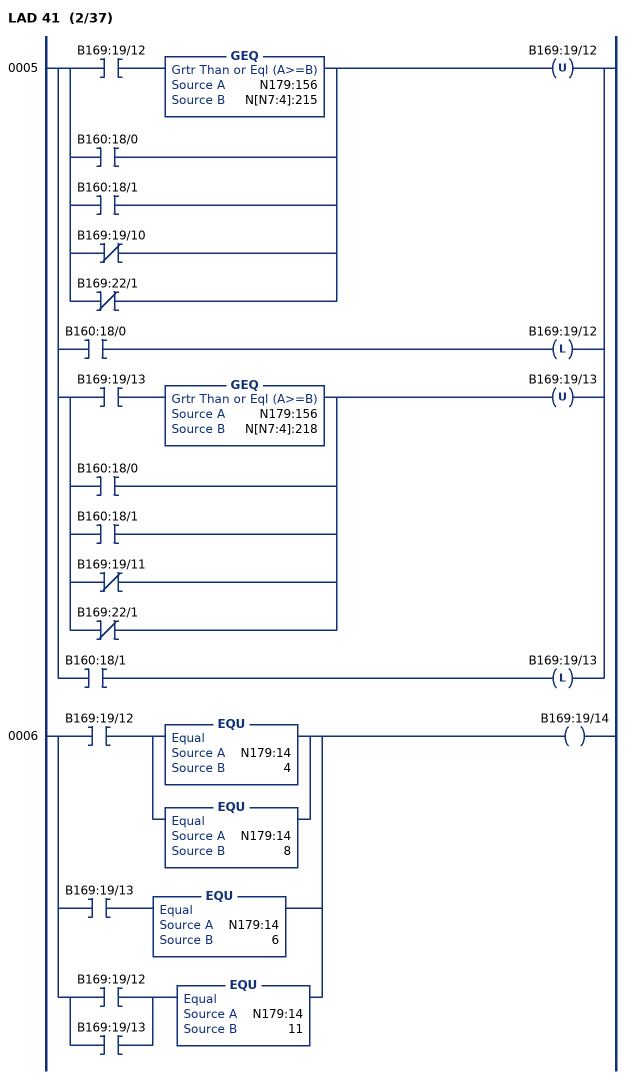
% Rung: 5 %
SOR BST BST BST XIC B169:19/12 GEQ N179:156 N[N7:4]:215 NXB BST XIC B160:18/0 NXB XIC B160:18/1 BND NXB XIO B169:19/10 NXB XIO B169:22/1 BND OTU B169:19/12 NXB XIC B160:18/0 OTL B169:19/12 BND NXB BST BST XIC B169:19/13 GEQ N179:156 N[N7:4]:218 NXB BST XIC B160:18/0 NXB XIC B160:18/1 BND NXB XIO B169:19/11 NXB XIO B169:22/1 BND OTU B169:19/13 NXB XIC B160:18/1 OTL B169:19/13 BND BND EOR
% Rung: 6 %
SOR BST XIC B169:19/12 BST EQU N179:14 4 NXB EQU N179:14 8 BND NXB XIC B169:19/13 EQU N179:14 6 NXB BST XIC B169:19/12 NXB XIC B169:19/13 BND EQU N179:14 11 BND OTE B169:19/14 EOR

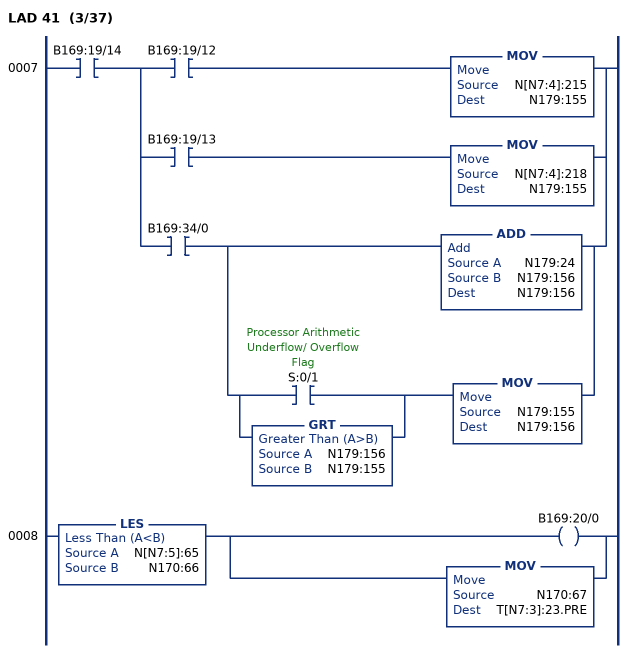
% Rung: 7 %
SOR XIC B169:19/14 BST BST XIC B169:19/12 MOV N[N7:4]:215 N179:155 NXB XIC B169:19/13 MOV N[N7:4]:218 N179:155 BND NXB XIC B169:34/0 BST ADD N179:24 N179:156 N179:156 NXB BST XIC S:0/1 NXB GRT N179:156 N179:155 BND MOV N179:155 N179:156 BND BND EOR
%   S:0/1  "Processor Arithmetic Underflow/ Overflow Flag" %
% Rung: 8 %
SOR LES N[N7:5]:65 N170:66 BST OTE B169:20/0 NXB MOV N170:67 T[N7:3]:23.PRE BND EOR

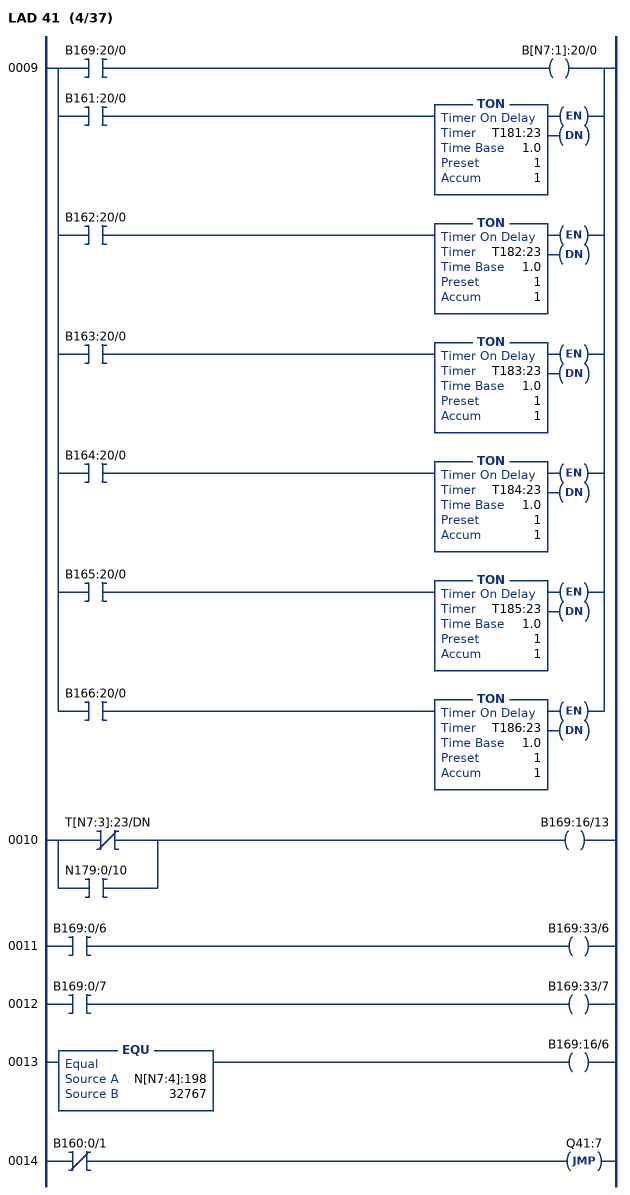
% Rung: 9 %
SOR BST XIC B169:20/0 OTE B[N7:1]:20/0 NXB XIC B161:20/0 TON T181:23 1.0 1 1 NXB XIC B162:20/0 TON T182:23 1.0 1 1 NXB XIC B163:20/0 TON T183:23 1.0 1 1 NXB XIC B164:20/0 TON T184:23 1.0 1 1 NXB XIC B165:20/0 TON T185:23 1.0 1 1 NXB XIC B166:20/0 TON T186:23 1.0 1 1 BND EOR
% Rung: 10 %
SOR BST XIO T[N7:3]:23/DN NXB XIC N179:0/10 BND OTE B169:16/13 EOR
% Rung: 11 %
SOR XIC B169:0/6 OTE B169:33/6 EOR
% Rung: 12 %
SOR XIC B169:0/7 OTE B169:33/7 EOR
% Rung: 13 %
SOR EQU N[N7:4]:198 32767 OTE B169:16/6 EOR
% Rung: 14 %
SOR XIO B160:0/1 JMP Q41:7 EOR

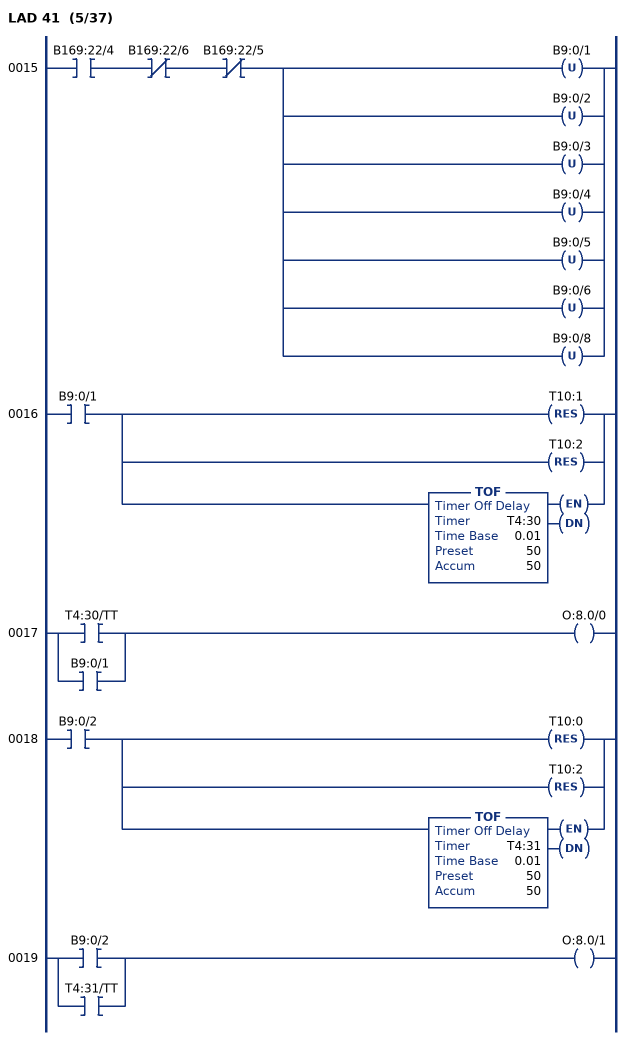
% Rung: 15 %
SOR XIC B169:22/4 XIO B169:22/6 XIO B169:22/5 BST OTU B9:0/1 NXB OTU B9:0/2 NXB OTU B9:0/3 NXB OTU B9:0/4 NXB OTU B9:0/5 NXB OTU B9:0/6 NXB OTU B9:0/8 BND EOR
% Rung: 16 %
SOR XIC B9:0/1 BST RES T10:1 NXB RES T10:2 NXB TOF T4:30 0.01 50 50 BND EOR
% Rung: 17 %
SOR BST XIC T4:30/TT NXB XIC B9:0/1 BND OTE O:8.0/0 EOR
% Rung: 18 %
SOR XIC B9:0/2 BST RES T10:0 NXB RES T10:2 NXB TOF T4:31 0.01 50 50 BND EOR
% Rung: 19 %
SOR BST XIC B9:0/2 NXB XIC T4:31/TT BND OTE O:8.0/1 EOR

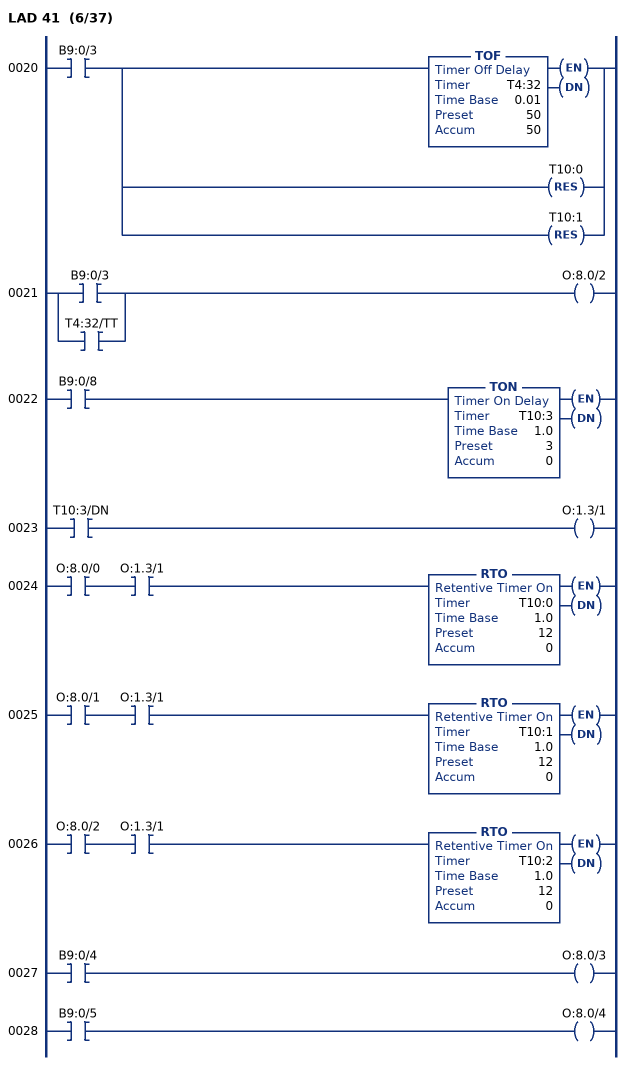
% Rung: 20 %
SOR XIC B9:0/3 BST TOF T4:32 0.01 50 50 NXB RES T10:0 NXB RES T10:1 BND EOR
% Rung: 21 %
SOR BST XIC B9:0/3 NXB XIC T4:32/TT BND OTE O:8.0/2 EOR
% Rung: 22 %
SOR XIC B9:0/8 TON T10:3 1.0 3 0 EOR
% Rung: 23 %
SOR XIC T10:3/DN OTE O:1.3/1 EOR
% Rung: 24 %
SOR XIC O:8.0/0 XIC O:1.3/1 RTO T10:0 1.0 12 0 EOR
% Rung: 25 %
SOR XIC O:8.0/1 XIC O:1.3/1 RTO T10:1 1.0 12 0 EOR
% Rung: 26 %
SOR XIC O:8.0/2 XIC O:1.3/1 RTO T10:2 1.0 12 0 EOR
% Rung: 27 %
SOR XIC B9:0/4 OTE O:8.0/3 EOR
% Rung: 28 %
SOR XIC B9:0/5 OTE O:8.0/4 EOR

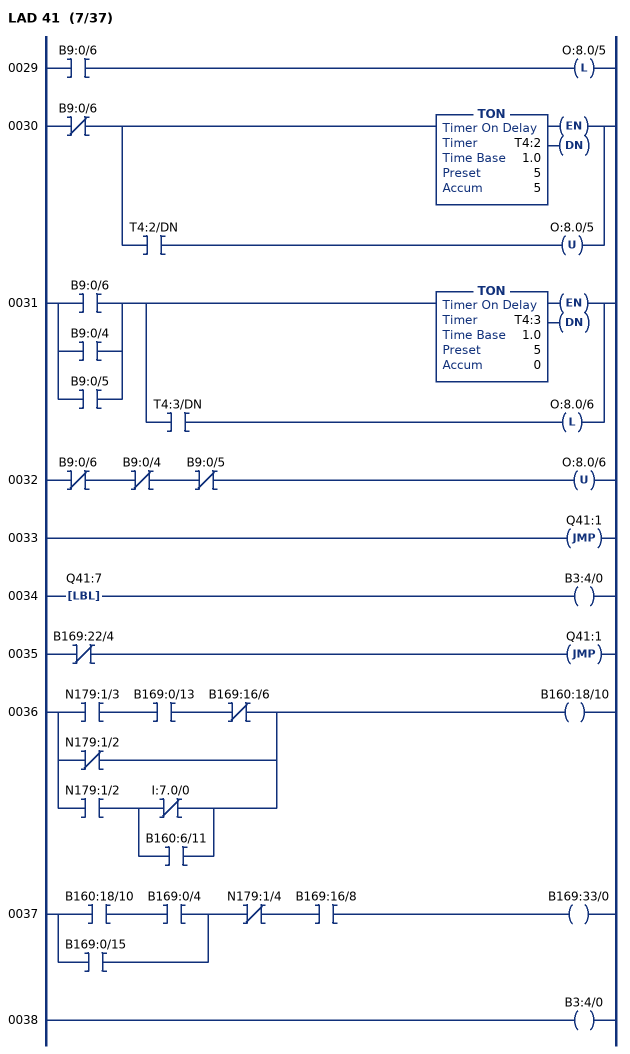
% Rung: 29 %
SOR XIC B9:0/6 OTL O:8.0/5 EOR
% Rung: 30 %
SOR XIO B9:0/6 BST TON T4:2 1.0 5 5 NXB XIC T4:2/DN OTU O:8.0/5 BND EOR
% Rung: 31 %
SOR BST XIC B9:0/6 NXB BST XIC B9:0/4 NXB XIC B9:0/5 BND BND BST TON T4:3 1.0 5 0 NXB XIC T4:3/DN OTL O:8.0/6 BND EOR
% Rung: 32 %
SOR XIO B9:0/6 XIO B9:0/4 XIO B9:0/5 OTU O:8.0/6 EOR
% Rung: 33 %
SOR JMP Q41:1 EOR
% Rung: 34 %
SOR LBL Q41:7 OTE B3:4/0 EOR
% Rung: 35 %
SOR XIO B169:22/4 JMP Q41:1 EOR
% Rung: 36 %
SOR BST XIC N179:1/3 XIC B169:0/13 XIO B169:16/6 NXB XIO N179:1/2 NXB XIC N179:1/2 BST XIO I:7.0/0 NXB XIC B160:6/11 BND BND OTE B160:18/10 EOR
% Rung: 37 %
SOR BST XIC B160:18/10 XIC B169:0/4 NXB XIC B169:0/15 BND XIO N179:1/4 XIC B169:16/8 OTE B169:33/0 EOR
% Rung: 38 %
SOR OTE B3:4/0 EOR

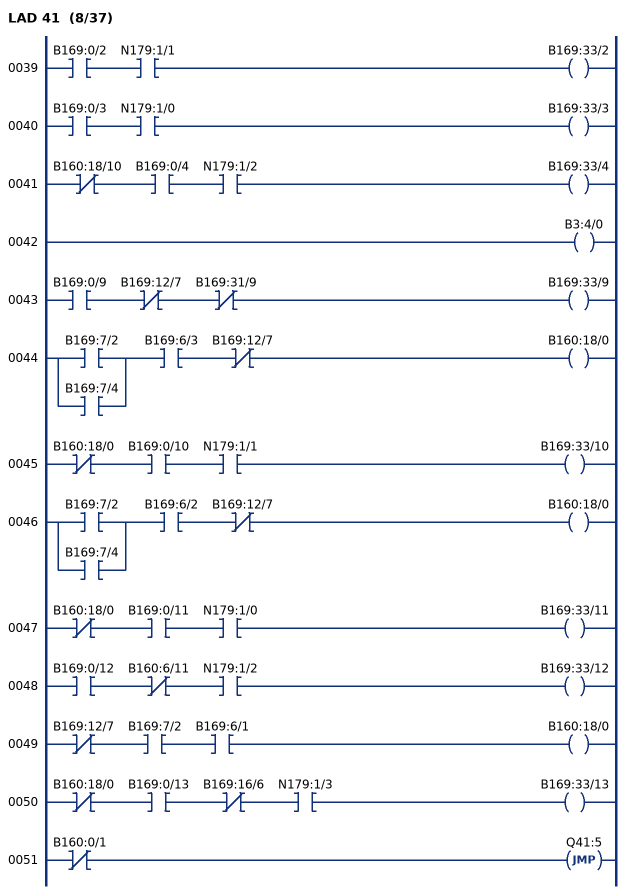
% Rung: 39 %
SOR XIC B169:0/2 XIC N179:1/1 OTE B169:33/2 EOR
% Rung: 40 %
SOR XIC B169:0/3 XIC N179:1/0 OTE B169:33/3 EOR
% Rung: 41 %
SOR XIO B160:18/10 XIC B169:0/4 XIC N179:1/2 OTE B169:33/4 EOR
% Rung: 42 %
SOR OTE B3:4/0 EOR
% Rung: 43 %
SOR XIC B169:0/9 XIO B169:12/7 XIO B169:31/9 OTE B169:33/9 EOR
% Rung: 44 %
SOR BST XIC B169:7/2 NXB XIC B169:7/4 BND XIC B169:6/3 XIO B169:12/7 OTE B160:18/0 EOR
% Rung: 45 %
SOR XIO B160:18/0 XIC B169:0/10 XIC N179:1/1 OTE B169:33/10 EOR
% Rung: 46 %
SOR BST XIC B169:7/2 NXB XIC B169:7/4 BND XIC B169:6/2 XIO B169:12/7 OTE B160:18/0 EOR
% Rung: 47 %
SOR XIO B160:18/0 XIC B169:0/11 XIC N179:1/0 OTE B169:33/11 EOR
% Rung: 48 %
SOR XIC B169:0/12 XIO B160:6/11 XIC N179:1/2 OTE B169:33/12 EOR
% Rung: 49 %
SOR XIO B169:12/7 XIC B169:7/2 XIC B169:6/1 OTE B160:18/0 EOR
% Rung: 50 %
SOR XIO B160:18/0 XIC B169:0/13 XIO B169:16/6 XIC N179:1/3 OTE B169:33/13 EOR
% Rung: 51 %
SOR XIO B160:0/1 JMP Q41:5 EOR

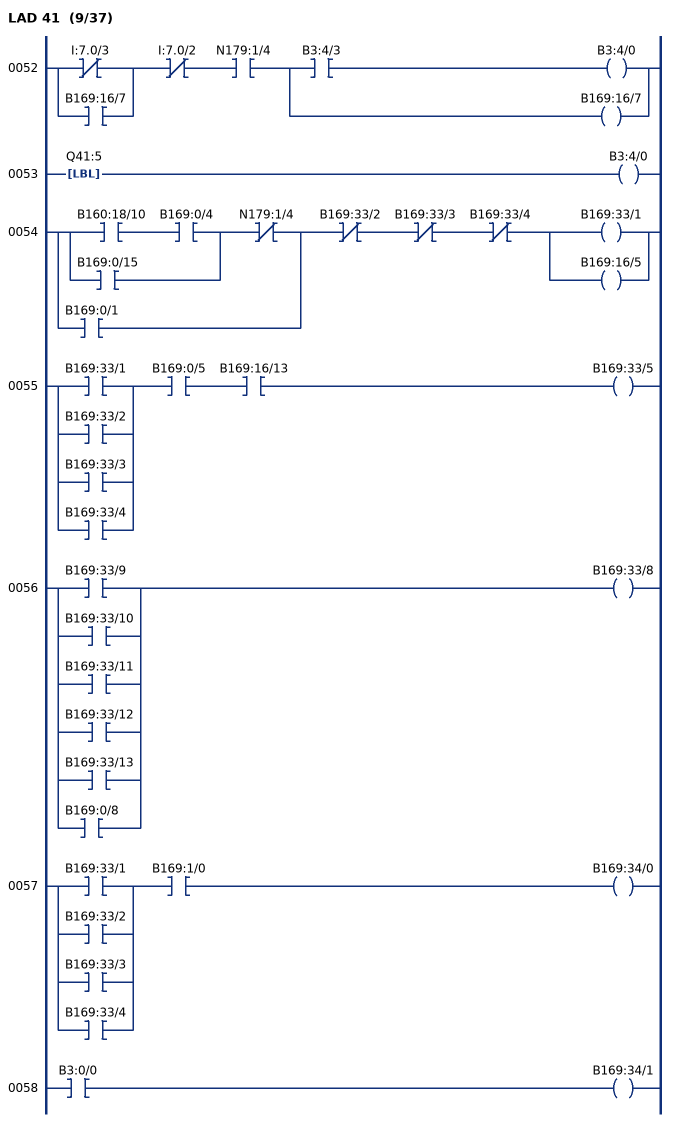
% Rung: 52 %
SOR BST XIO I:7.0/3 NXB XIC B169:16/7 BND XIO I:7.0/2 XIC N179:1/4 BST XIC B3:4/3 OTE B3:4/0 NXB OTE B169:16/7 BND EOR
% Rung: 53 %
SOR LBL Q41:5 OTE B3:4/0 EOR
% Rung: 54 %
SOR BST BST XIC B160:18/10 XIC B169:0/4 NXB XIC B169:0/15 BND XIO N179:1/4 NXB XIC B169:0/1 BND XIO B169:33/2 XIO B169:33/3 XIO B169:33/4 BST OTE B169:33/1 NXB OTE B169:16/5 BND EOR
% Rung: 55 %
SOR BST XIC B169:33/1 NXB XIC B169:33/2 NXB XIC B169:33/3 NXB XIC B169:33/4 BND XIC B169:0/5 XIC B169:16/13 OTE B169:33/5 EOR
% Rung: 56 %
SOR BST XIC B169:33/9 NXB XIC B169:33/10 NXB XIC B169:33/11 NXB XIC B169:33/12 NXB XIC B169:33/13 NXB XIC B169:0/8 BND OTE B169:33/8 EOR
% Rung: 57 %
SOR BST XIC B169:33/1 NXB XIC B169:33/2 NXB XIC B169:33/3 NXB XIC B169:33/4 BND XIC B169:1/0 OTE B169:34/0 EOR
% Rung: 58 %
SOR XIC B3:0/0 OTE B169:34/1 EOR

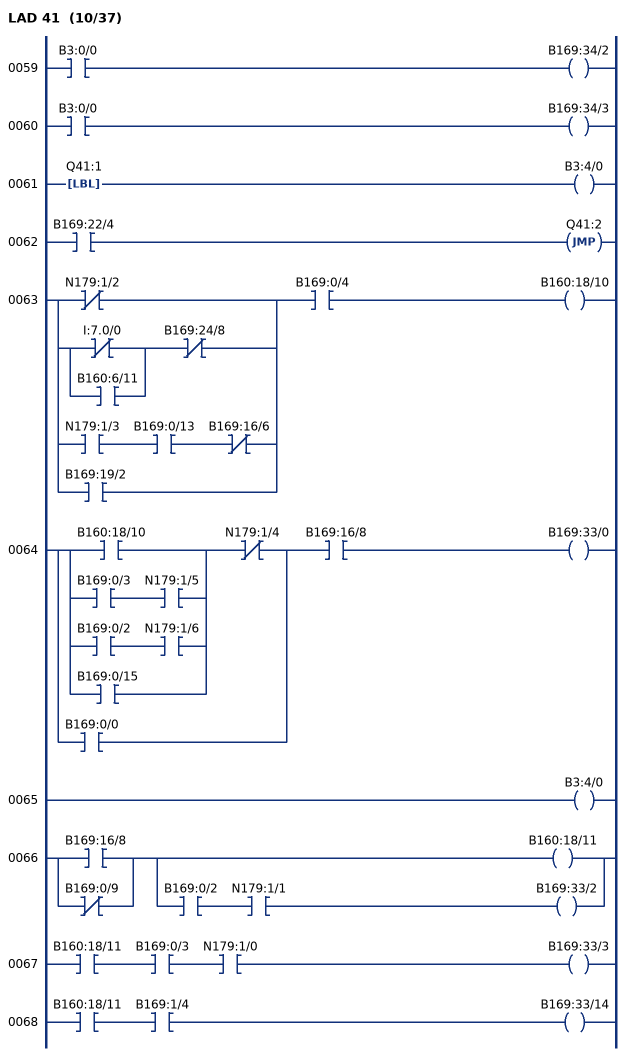
% Rung: 59 %
SOR XIC B3:0/0 OTE B169:34/2 EOR
% Rung: 60 %
SOR XIC B3:0/0 OTE B169:34/3 EOR
% Rung: 61 %
SOR LBL Q41:1 OTE B3:4/0 EOR
% Rung: 62 %
SOR XIC B169:22/4 JMP Q41:2 EOR
% Rung: 63 %
SOR BST XIO N179:1/2 NXB BST XIO I:7.0/0 NXB XIC B160:6/11 BND XIO B169:24/8 NXB XIC N179:1/3 XIC B169:0/13 XIO B169:16/6 NXB XIC B169:19/2 BND XIC B169:0/4 OTE B160:18/10 EOR
% Rung: 64 %
SOR BST BST XIC B160:18/10 NXB XIC B169:0/3 XIC N179:1/5 NXB XIC B169:0/2 XIC N179:1/6 NXB XIC B169:0/15 BND XIO N179:1/4 NXB XIC B169:0/0 BND XIC B169:16/8 OTE B169:33/0 EOR
% Rung: 65 %
SOR OTE B3:4/0 EOR
% Rung: 66 %
SOR BST XIC B169:16/8 NXB XIO B169:0/9 BND BST OTE B160:18/11 NXB XIC B169:0/2 XIC N179:1/1 OTE B169:33/2 BND EOR
% Rung: 67 %
SOR XIC B160:18/11 XIC B169:0/3 XIC N179:1/0 OTE B169:33/3 EOR
% Rung: 68 %
SOR XIC B160:18/11 XIC B169:1/4 OTE B169:33/14 EOR

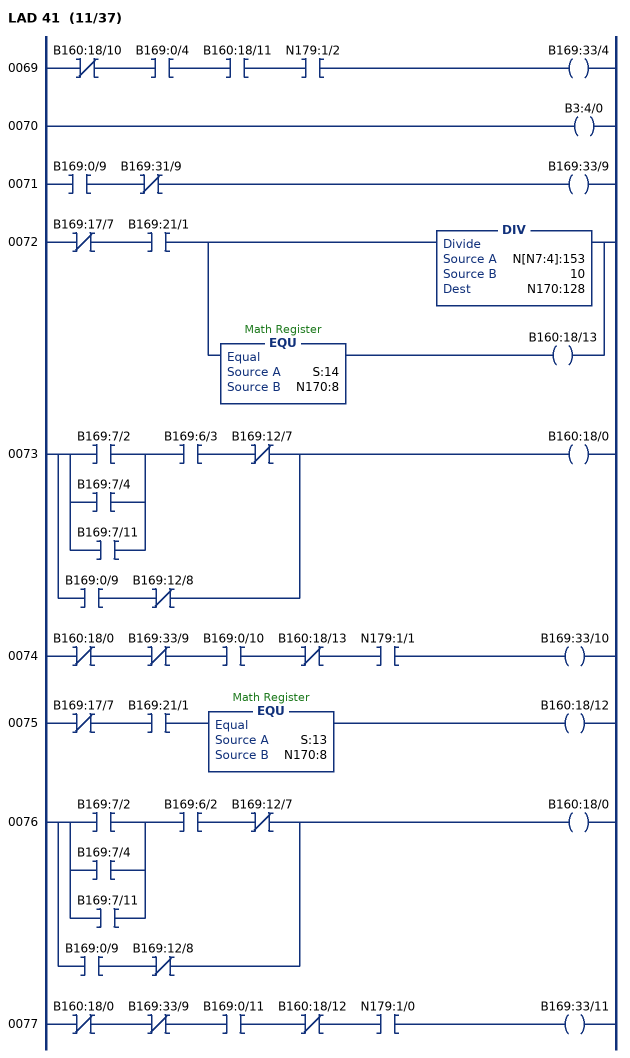
% Rung: 69 %
SOR XIO B160:18/10 XIC B169:0/4 XIC B160:18/11 XIC N179:1/2 OTE B169:33/4 EOR
% Rung: 70 %
SOR OTE B3:4/0 EOR
% Rung: 71 %
SOR XIC B169:0/9 XIO B169:31/9 OTE B169:33/9 EOR
% Rung: 72 %
SOR XIO B169:17/7 XIC B169:21/1 BST DIV N[N7:4]:153 10 N170:128 NXB EQU S:14 N170:8 OTE B160:18/13 BND EOR
%   S:14  "Math Register" %
% Rung: 73 %
SOR BST BST XIC B169:7/2 NXB XIC B169:7/4 NXB XIC B169:7/11 BND XIC B169:6/3 XIO B169:12/7 NXB XIC B169:0/9 XIO B169:12/8 BND OTE B160:18/0 EOR
% Rung: 74 %
SOR XIO B160:18/0 XIO B169:33/9 XIC B169:0/10 XIO B160:18/13 XIC N179:1/1 OTE B169:33/10 EOR
% Rung: 75 %
SOR XIO B169:17/7 XIC B169:21/1 EQU S:13 N170:8 OTE B160:18/12 EOR
%   S:13  "Math Register" %
% Rung: 76 %
SOR BST BST XIC B169:7/2 NXB XIC B169:7/4 NXB XIC B169:7/11 BND XIC B169:6/2 XIO B169:12/7 NXB XIC B169:0/9 XIO B169:12/8 BND OTE B160:18/0 EOR
% Rung: 77 %
SOR XIO B160:18/0 XIO B169:33/9 XIC B169:0/11 XIO B160:18/12 XIC N179:1/0 OTE B169:33/11 EOR

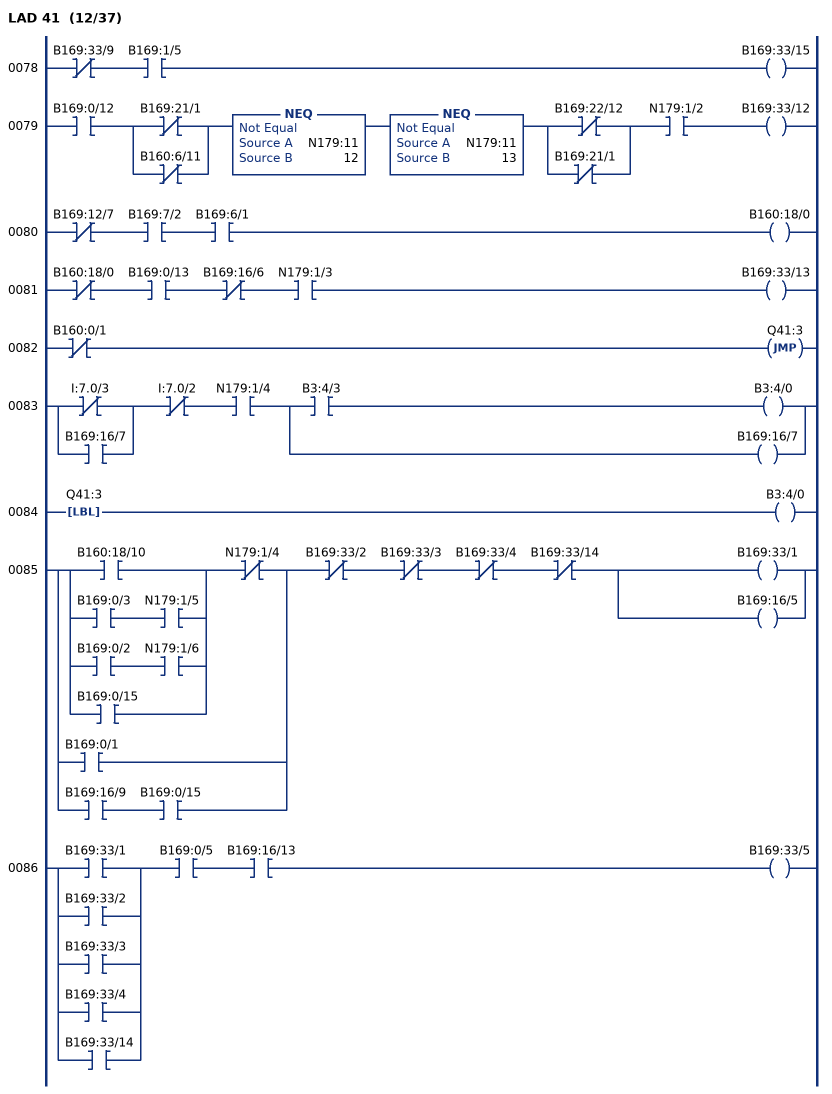
% Rung: 78 %
SOR XIO B169:33/9 XIC B169:1/5 OTE B169:33/15 EOR
% Rung: 79 %
SOR XIC B169:0/12 BST XIO B169:21/1 NXB XIO B160:6/11 BND NEQ N179:11 12 NEQ N179:11 13 BST XIO B169:22/12 NXB XIO B169:21/1 BND XIC N179:1/2 OTE B169:33/12 EOR
% Rung: 80 %
SOR XIO B169:12/7 XIC B169:7/2 XIC B169:6/1 OTE B160:18/0 EOR
% Rung: 81 %
SOR XIO B160:18/0 XIC B169:0/13 XIO B169:16/6 XIC N179:1/3 OTE B169:33/13 EOR
% Rung: 82 %
SOR XIO B160:0/1 JMP Q41:3 EOR
% Rung: 83 %
SOR BST XIO I:7.0/3 NXB XIC B169:16/7 BND XIO I:7.0/2 XIC N179:1/4 BST XIC B3:4/3 OTE B3:4/0 NXB OTE B169:16/7 BND EOR
% Rung: 84 %
SOR LBL Q41:3 OTE B3:4/0 EOR
% Rung: 85 %
SOR BST BST XIC B160:18/10 NXB XIC B169:0/3 XIC N179:1/5 NXB XIC B169:0/2 XIC N179:1/6 NXB XIC B169:0/15 BND XIO N179:1/4 NXB XIC B169:0/1 NXB XIC B169:16/9 XIC B169:0/15 BND XIO B169:33/2 XIO B169:33/3 XIO B169:33/4 XIO B169:33/14 BST OTE B169:33/1 NXB OTE B169:16/5 BND EOR
% Rung: 86 %
SOR BST XIC B169:33/1 NXB XIC B169:33/2 NXB XIC B169:33/3 NXB XIC B169:33/4 NXB XIC B169:33/14 BND XIC B169:0/5 XIC B169:16/13 OTE B169:33/5 EOR

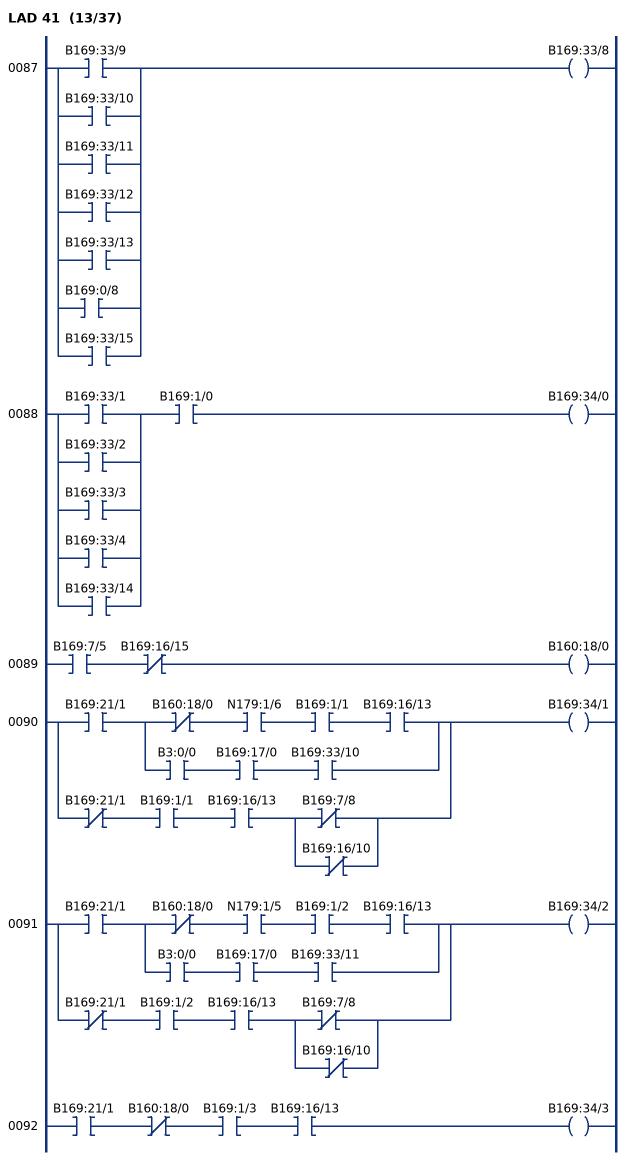
% Rung: 87 %
SOR BST XIC B169:33/9 NXB XIC B169:33/10 NXB XIC B169:33/11 NXB XIC B169:33/12 NXB XIC B169:33/13 NXB XIC B169:0/8 NXB XIC B169:33/15 BND OTE B169:33/8 EOR
% Rung: 88 %
SOR BST XIC B169:33/1 NXB XIC B169:33/2 NXB XIC B169:33/3 NXB XIC B169:33/4 NXB XIC B169:33/14 BND XIC B169:1/0 OTE B169:34/0 EOR
% Rung: 89 %
SOR XIC B169:7/5 XIO B169:16/15 OTE B160:18/0 EOR
% Rung: 90 %
SOR BST XIC B169:21/1 BST XIO B160:18/0 XIC N179:1/6 XIC B169:1/1 XIC B169:16/13 NXB XIC B3:0/0 XIC B169:17/0 XIC B169:33/10 BND NXB XIO B169:21/1 XIC B169:1/1 XIC B169:16/13 BST XIO B169:7/8 NXB XIO B169:16/10 BND BND OTE B169:34/1 EOR
% Rung: 91 %
SOR BST XIC B169:21/1 BST XIO B160:18/0 XIC N179:1/5 XIC B169:1/2 XIC B169:16/13 NXB XIC B3:0/0 XIC B169:17/0 XIC B169:33/11 BND NXB XIO B169:21/1 XIC B169:1/2 XIC B169:16/13 BST XIO B169:7/8 NXB XIO B169:16/10 BND BND OTE B169:34/2 EOR
% Rung: 92 %
SOR XIC B169:21/1 XIO B160:18/0 XIC B169:1/3 XIC B169:16/13 OTE B169:34/3 EOR

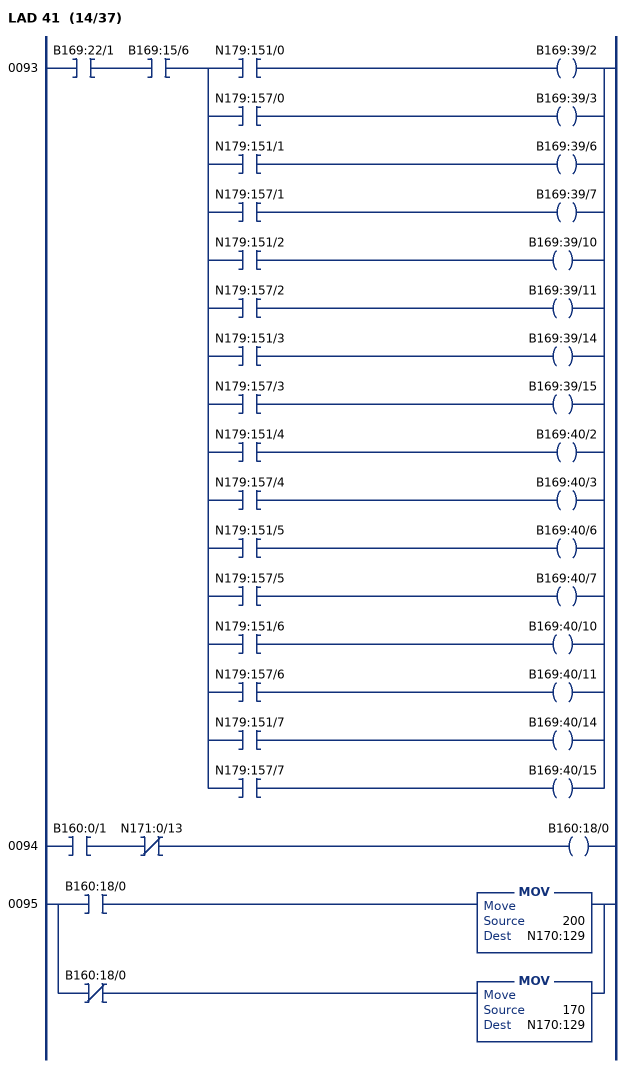
% Rung: 93 %
SOR XIC B169:22/1 XIC B169:15/6 BST BST XIC N179:151/0 OTE B169:39/2 NXB XIC N179:157/0 OTE B169:39/3 BND NXB BST XIC N179:151/1 OTE B169:39/6 NXB XIC N179:157/1 OTE B169:39/7 BND NXB BST XIC N179:151/2 OTE B169:39/10 NXB XIC N179:157/2 OTE B169:39/11 BND NXB BST XIC N179:151/3 OTE B169:39/14 NXB XIC N179:157/3 OTE B169:39/15 BND NXB BST XIC N179:151/4 OTE B169:40/2 NXB XIC N179:157/4 OTE B169:40/3 BND NXB BST XIC N179:151/5 OTE B169:40/6 NXB XIC N179:157/5 OTE B169:40/7 BND NXB BST XIC N179:151/6 OTE B169:40/10 NXB XIC N179:157/6 OTE B169:40/11 BND NXB BST XIC N179:151/7 OTE B169:40/14 NXB XIC N179:157/7 OTE B169:40/15 BND BND EOR
% Rung: 94 %
SOR XIC B160:0/1 XIO N171:0/13 OTE B160:18/0 EOR
% Rung: 95 %
SOR BST XIC B160:18/0 MOV 200 N170:129 NXB XIO B160:18/0 MOV 170 N170:129 BND EOR

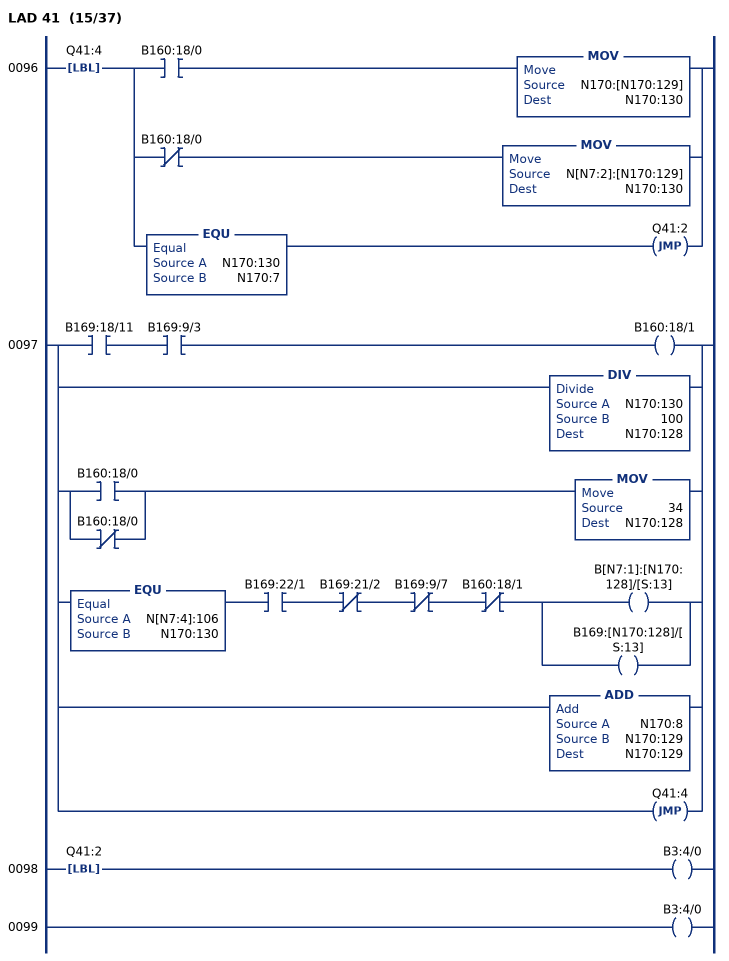
% Rung: 96 %
SOR LBL Q41:4 BST XIC B160:18/0 MOV N170:[N170:129] N170:130 NXB XIO B160:18/0 MOV N[N7:2]:[N170:129] N170:130 NXB EQU N170:130 N170:7 JMP Q41:2 BND EOR
% Rung: 97 %
SOR BST XIC B169:18/11 XIC B169:9/3 OTE B160:18/1 NXB BST DIV N170:130 100 N170:128 NXB BST XIC B160:18/0 NXB XIO B160:18/0 BND MOV 34 N170:128 NXB EQU N[N7:4]:106 N170:130 XIC B169:22/1 XIO B169:21/2 XIO B169:9/7 XIO B160:18/1 BST OTE B[N7:1]:[N170:128]/[S:13] NXB OTE B169:[N170:128]/[S:13] BND BND NXB ADD N170:8 N170:129 N170:129 NXB JMP Q41:4 BND EOR
%   S:13  "Math Register" %
% Rung: 98 %
SOR LBL Q41:2 OTE B3:4/0 EOR
% Rung: 99 %
SOR OTE B3:4/0 EOR

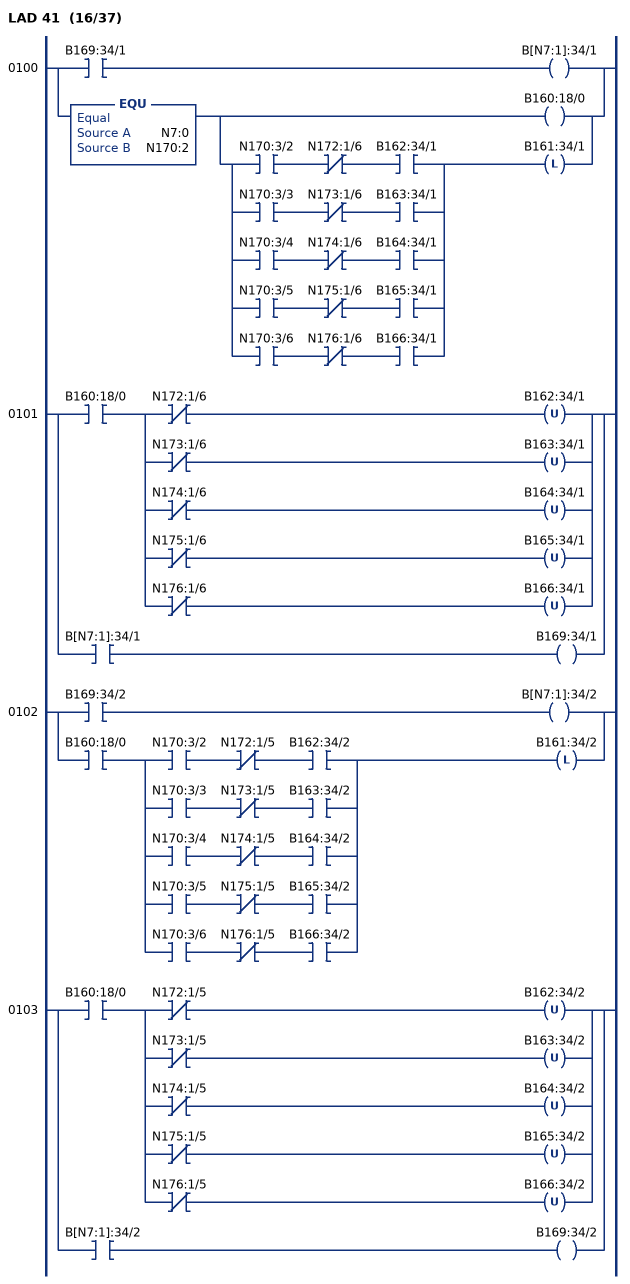
% Rung: 100 %
SOR BST XIC B169:34/1 OTE B[N7:1]:34/1 NXB EQU N7:0 N170:2 BST OTE B160:18/0 NXB BST XIC N170:3/2 XIO N172:1/6 XIC B162:34/1 NXB XIC N170:3/3 XIO N173:1/6 XIC B163:34/1 NXB XIC N170:3/4 XIO N174:1/6 XIC B164:34/1 NXB XIC N170:3/5 XIO N175:1/6 XIC B165:34/1 NXB XIC N170:3/6 XIO N176:1/6 XIC B166:34/1 BND OTL B161:34/1 BND BND EOR
% Rung: 101 %
SOR BST XIC B160:18/0 BST XIO N172:1/6 OTU B162:34/1 NXB XIO N173:1/6 OTU B163:34/1 NXB XIO N174:1/6 OTU B164:34/1 NXB XIO N175:1/6 OTU B165:34/1 NXB XIO N176:1/6 OTU B166:34/1 BND NXB XIC B[N7:1]:34/1 OTE B169:34/1 BND EOR
% Rung: 102 %
SOR BST XIC B169:34/2 OTE B[N7:1]:34/2 NXB XIC B160:18/0 BST XIC N170:3/2 XIO N172:1/5 XIC B162:34/2 NXB XIC N170:3/3 XIO N173:1/5 XIC B163:34/2 NXB XIC N170:3/4 XIO N174:1/5 XIC B164:34/2 NXB XIC N170:3/5 XIO N175:1/5 XIC B165:34/2 NXB XIC N170:3/6 XIO N176:1/5 XIC B166:34/2 BND OTL B161:34/2 BND EOR
% Rung: 103 %
SOR BST XIC B160:18/0 BST XIO N172:1/5 OTU B162:34/2 NXB XIO N173:1/5 OTU B163:34/2 NXB XIO N174:1/5 OTU B164:34/2 NXB XIO N175:1/5 OTU B165:34/2 NXB XIO N176:1/5 OTU B166:34/2 BND NXB XIC B[N7:1]:34/2 OTE B169:34/2 BND EOR

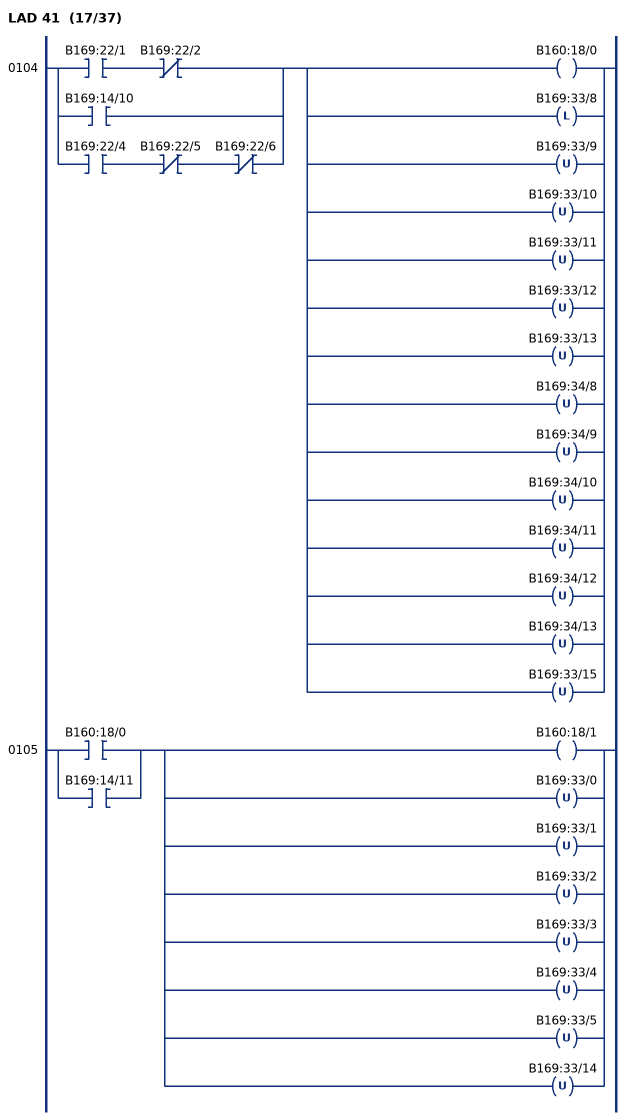
% Rung: 104 %
SOR BST XIC B169:22/1 XIO B169:22/2 NXB XIC B169:14/10 NXB XIC B169:22/4 XIO B169:22/5 XIO B169:22/6 BND BST OTE B160:18/0 NXB OTL B169:33/8 NXB OTU B169:33/9 NXB OTU B169:33/10 NXB OTU B169:33/11 NXB OTU B169:33/12 NXB OTU B169:33/13 NXB OTU B169:34/8 NXB OTU B169:34/9 NXB OTU B169:34/10 NXB OTU B169:34/11 NXB OTU B169:34/12 NXB OTU B169:34/13 NXB OTU B169:33/15 BND EOR
% Rung: 105 %
SOR BST XIC B160:18/0 NXB XIC B169:14/11 BND BST OTE B160:18/1 NXB OTU B169:33/0 NXB OTU B169:33/1 NXB OTU B169:33/2 NXB OTU B169:33/3 NXB OTU B169:33/4 NXB OTU B169:33/5 NXB OTU B169:33/14 BND EOR

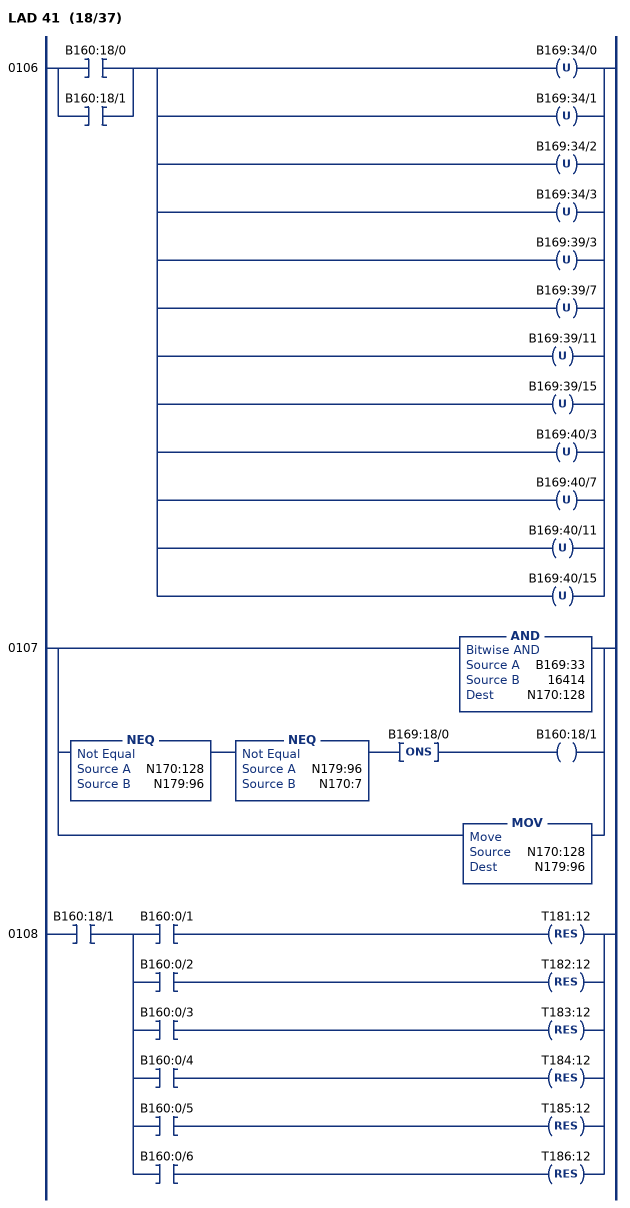
% Rung: 106 %
SOR BST XIC B160:18/0 NXB XIC B160:18/1 BND BST OTU B169:34/0 NXB OTU B169:34/1 NXB OTU B169:34/2 NXB OTU B169:34/3 NXB OTU B169:39/3 NXB OTU B169:39/7 NXB OTU B169:39/11 NXB OTU B169:39/15 NXB OTU B169:40/3 NXB OTU B169:40/7 NXB OTU B169:40/11 NXB OTU B169:40/15 BND EOR
% Rung: 107 %
SOR BST AND B169:33 16414 N170:128 NXB NEQ N170:128 N179:96 NEQ N179:96 N170:7 OSR B169:18/0 OTE B160:18/1 NXB MOV N170:128 N179:96 BND EOR
% Rung: 108 %
SOR XIC B160:18/1 BST XIC B160:0/1 RES T181:12 NXB XIC B160:0/2 RES T182:12 NXB XIC B160:0/3 RES T183:12 NXB XIC B160:0/4 RES T184:12 NXB XIC B160:0/5 RES T185:12 NXB XIC B160:0/6 RES T186:12 BND EOR

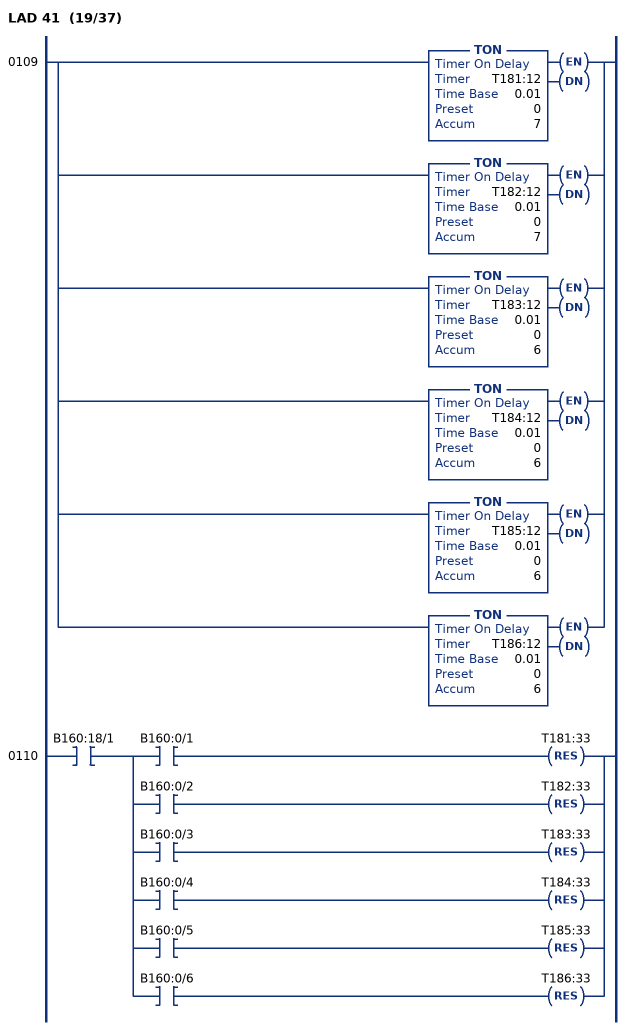
% Rung: 109 %
SOR BST TON T181:12 0.01 0 7 NXB TON T182:12 0.01 0 7 NXB TON T183:12 0.01 0 6 NXB TON T184:12 0.01 0 6 NXB TON T185:12 0.01 0 6 NXB TON T186:12 0.01 0 6 BND EOR
% Rung: 110 %
SOR XIC B160:18/1 BST XIC B160:0/1 RES T181:33 NXB XIC B160:0/2 RES T182:33 NXB XIC B160:0/3 RES T183:33 NXB XIC B160:0/4 RES T184:33 NXB XIC B160:0/5 RES T185:33 NXB XIC B160:0/6 RES T186:33 BND EOR

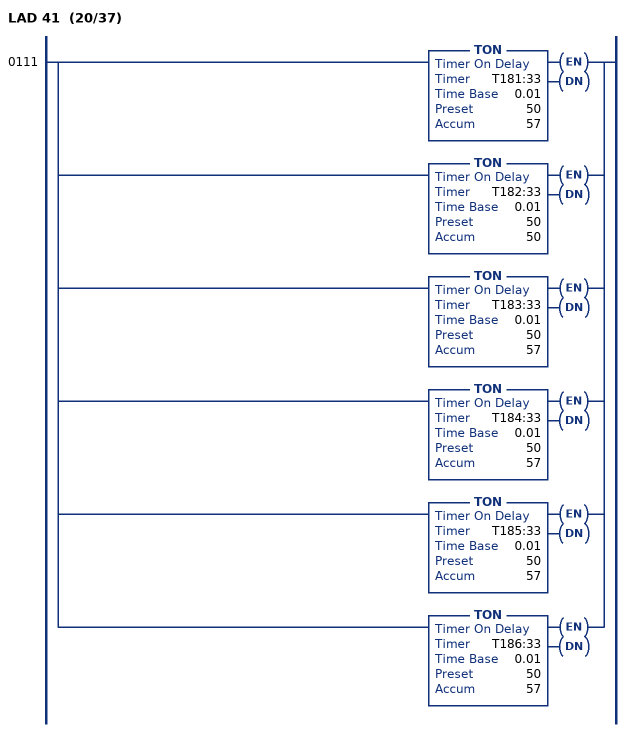
% Rung: 111 %
SOR BST TON T181:33 0.01 50 57 NXB TON T182:33 0.01 50 50 NXB TON T183:33 0.01 50 57 NXB TON T184:33 0.01 50 57 NXB TON T185:33 0.01 50 57 NXB TON T186:33 0.01 50 57 BND EOR

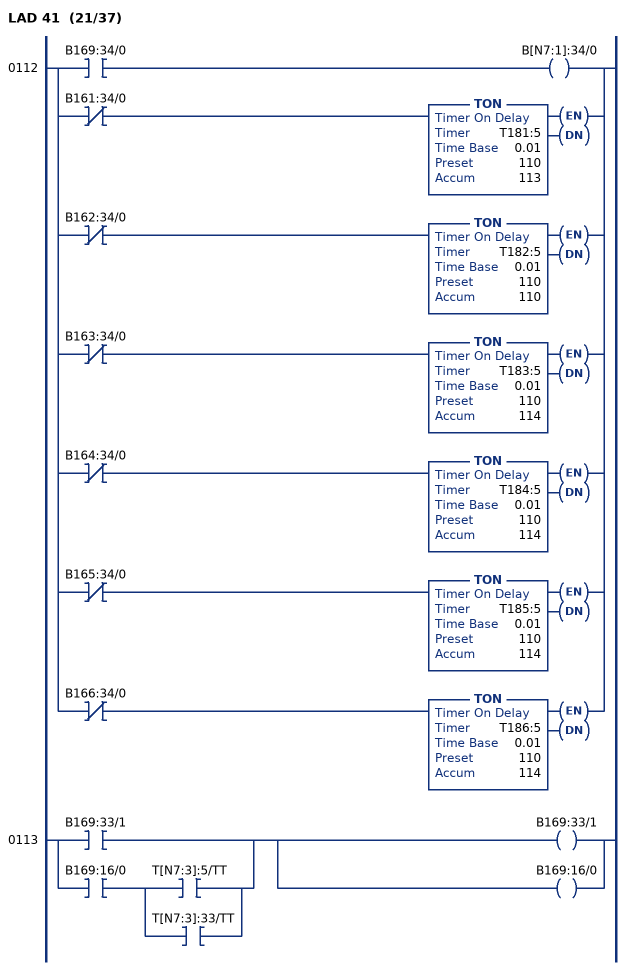
% Rung: 112 %
SOR BST XIC B169:34/0 OTE B[N7:1]:34/0 NXB XIO B161:34/0 TON T181:5 0.01 110 113 NXB XIO B162:34/0 TON T182:5 0.01 110 110 NXB XIO B163:34/0 TON T183:5 0.01 110 114 NXB XIO B164:34/0 TON T184:5 0.01 110 114 NXB XIO B165:34/0 TON T185:5 0.01 110 114 NXB XIO B166:34/0 TON T186:5 0.01 110 114 BND EOR
% Rung: 113 %
SOR BST XIC B169:33/1 NXB XIC B169:16/0 BST XIC T[N7:3]:5/TT NXB XIC T[N7:3]:33/TT BND BND BST OTE B169:33/1 NXB OTE B169:16/0 BND EOR

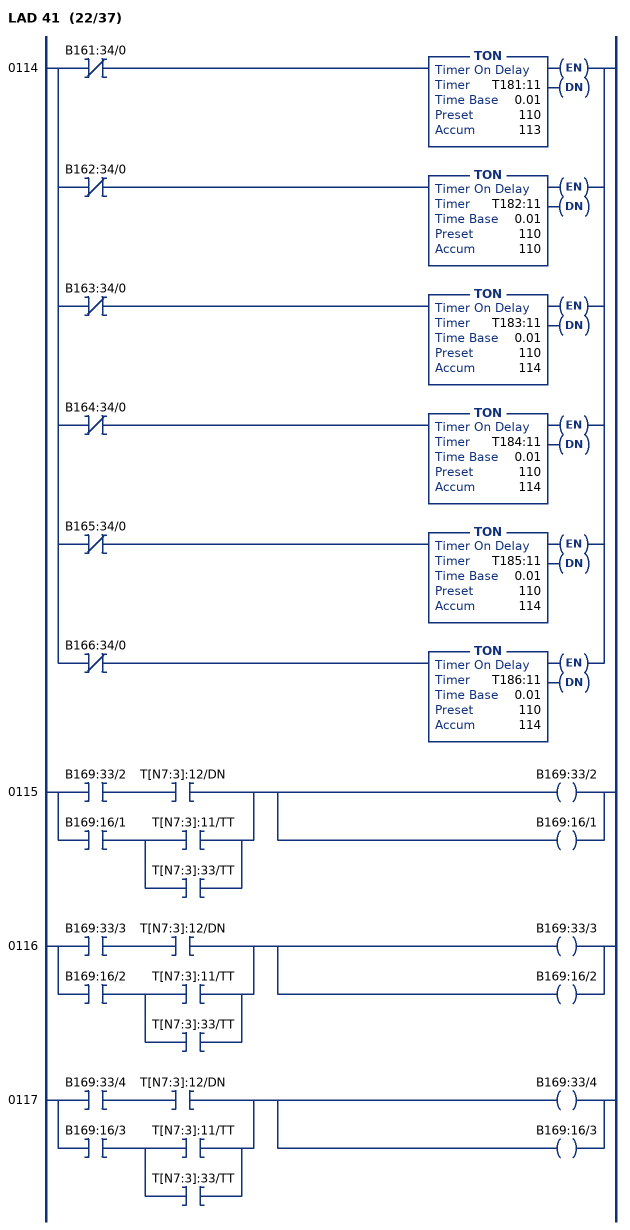
% Rung: 114 %
SOR BST XIO B161:34/0 TON T181:11 0.01 110 113 NXB XIO B162:34/0 TON T182:11 0.01 110 110 NXB XIO B163:34/0 TON T183:11 0.01 110 114 NXB XIO B164:34/0 TON T184:11 0.01 110 114 NXB XIO B165:34/0 TON T185:11 0.01 110 114 NXB XIO B166:34/0 TON T186:11 0.01 110 114 BND EOR
% Rung: 115 %
SOR BST XIC B169:33/2 XIC T[N7:3]:12/DN NXB XIC B169:16/1 BST XIC T[N7:3]:11/TT NXB XIC T[N7:3]:33/TT BND BND BST OTE B169:33/2 NXB OTE B169:16/1 BND EOR
% Rung: 116 %
SOR BST XIC B169:33/3 XIC T[N7:3]:12/DN NXB XIC B169:16/2 BST XIC T[N7:3]:11/TT NXB XIC T[N7:3]:33/TT BND BND BST OTE B169:33/3 NXB OTE B169:16/2 BND EOR
% Rung: 117 %
SOR BST XIC B169:33/4 XIC T[N7:3]:12/DN NXB XIC B169:16/3 BST XIC T[N7:3]:11/TT NXB XIC T[N7:3]:33/TT BND BND BST OTE B169:33/4 NXB OTE B169:16/3 BND EOR

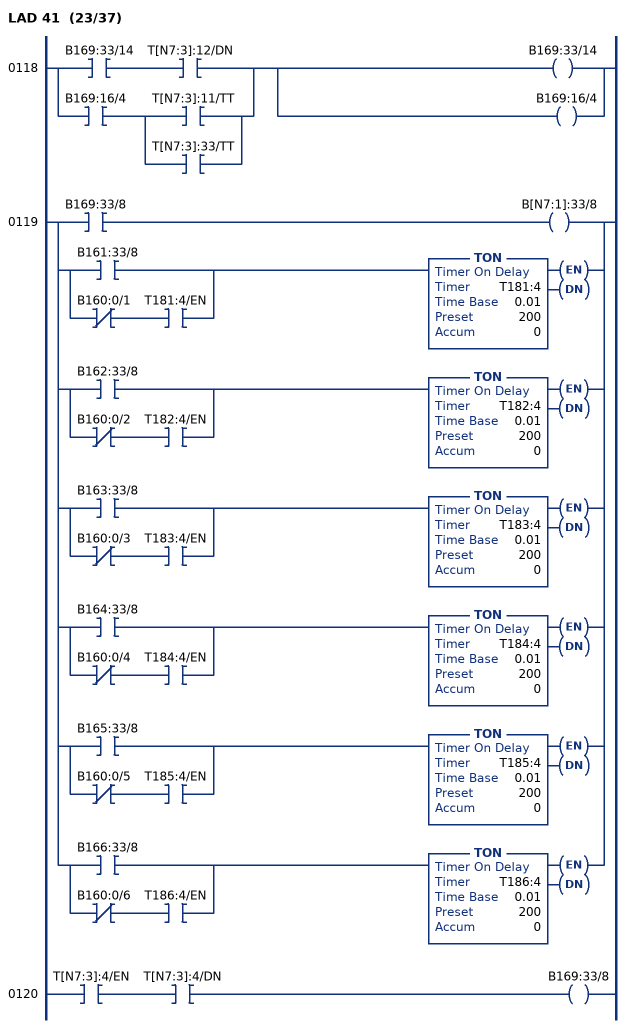
% Rung: 118 %
SOR BST XIC B169:33/14 XIC T[N7:3]:12/DN NXB XIC B169:16/4 BST XIC T[N7:3]:11/TT NXB XIC T[N7:3]:33/TT BND BND BST OTE B169:33/14 NXB OTE B169:16/4 BND EOR
% Rung: 119 %
SOR BST XIC B169:33/8 OTE B[N7:1]:33/8 NXB BST XIC B161:33/8 NXB XIO B160:0/1 XIC T181:4/EN BND TON T181:4 0.01 200 0 NXB BST XIC B162:33/8 NXB XIO B160:0/2 XIC T182:4/EN BND TON T182:4 0.01 200 0 NXB BST XIC B163:33/8 NXB XIO B160:0/3 XIC T183:4/EN BND TON T183:4 0.01 200 0 NXB BST XIC B164:33/8 NXB XIO B160:0/4 XIC T184:4/EN BND TON T184:4 0.01 200 0 NXB BST XIC B165:33/8 NXB XIO B160:0/5 XIC T185:4/EN BND TON T185:4 0.01 200 0 NXB BST XIC B166:33/8 NXB XIO B160:0/6 XIC T186:4/EN BND TON T186:4 0.01 200 0 BND EOR
% Rung: 120 %
SOR XIC T[N7:3]:4/EN XIC T[N7:3]:4/DN OTE B169:33/8 EOR

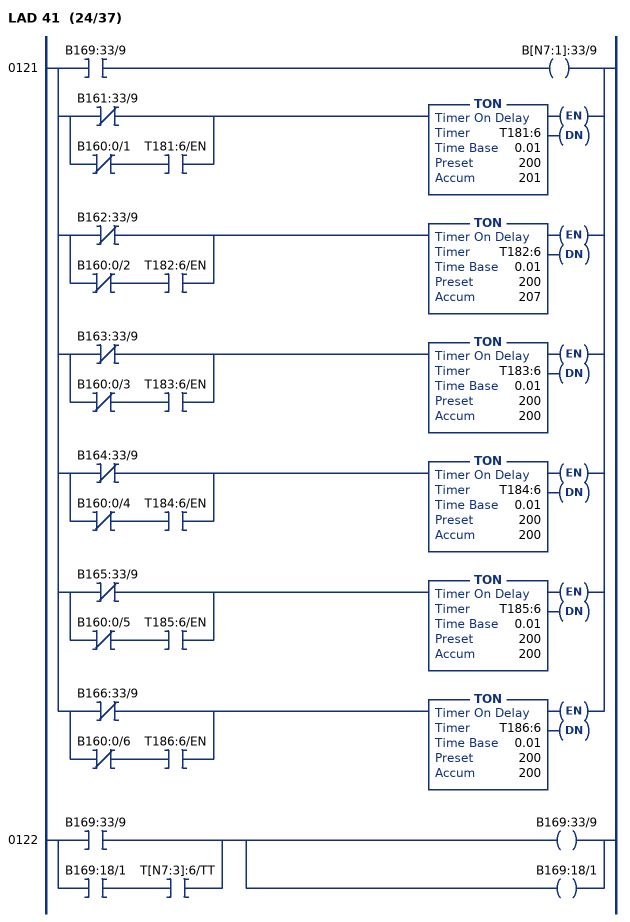
% Rung: 121 %
SOR BST XIC B169:33/9 OTE B[N7:1]:33/9 NXB BST XIO B161:33/9 NXB XIO B160:0/1 XIC T181:6/EN BND TON T181:6 0.01 200 201 NXB BST XIO B162:33/9 NXB XIO B160:0/2 XIC T182:6/EN BND TON T182:6 0.01 200 207 NXB BST XIO B163:33/9 NXB XIO B160:0/3 XIC T183:6/EN BND TON T183:6 0.01 200 200 NXB BST XIO B164:33/9 NXB XIO B160:0/4 XIC T184:6/EN BND TON T184:6 0.01 200 200 NXB BST XIO B165:33/9 NXB XIO B160:0/5 XIC T185:6/EN BND TON T185:6 0.01 200 200 NXB BST XIO B166:33/9 NXB XIO B160:0/6 XIC T186:6/EN BND TON T186:6 0.01 200 200 BND EOR
% Rung: 122 %
SOR BST XIC B169:33/9 NXB XIC B169:18/1 XIC T[N7:3]:6/TT BND BST OTE B169:33/9 NXB OTE B169:18/1 BND EOR

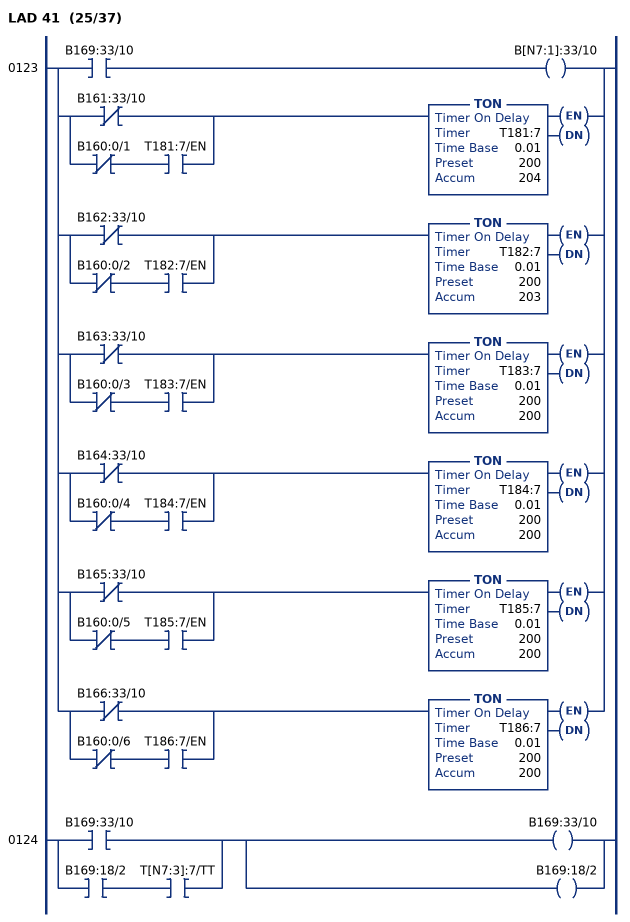
% Rung: 123 %
SOR BST XIC B169:33/10 OTE B[N7:1]:33/10 NXB BST XIO B161:33/10 NXB XIO B160:0/1 XIC T181:7/EN BND TON T181:7 0.01 200 204 NXB BST XIO B162:33/10 NXB XIO B160:0/2 XIC T182:7/EN BND TON T182:7 0.01 200 203 NXB BST XIO B163:33/10 NXB XIO B160:0/3 XIC T183:7/EN BND TON T183:7 0.01 200 200 NXB BST XIO B164:33/10 NXB XIO B160:0/4 XIC T184:7/EN BND TON T184:7 0.01 200 200 NXB BST XIO B165:33/10 NXB XIO B160:0/5 XIC T185:7/EN BND TON T185:7 0.01 200 200 NXB BST XIO B166:33/10 NXB XIO B160:0/6 XIC T186:7/EN BND TON T186:7 0.01 200 200 BND EOR
% Rung: 124 %
SOR BST XIC B169:33/10 NXB XIC B169:18/2 XIC T[N7:3]:7/TT BND BST OTE B169:33/10 NXB OTE B169:18/2 BND EOR

